FUNCTION_BLOCK DSInterface (* Drill station service interface *)
  (* Standard: 61499-2 *)
  (* Version 0.2, 2003-12-04, JHC, Rockwell Automation, Renamed for better indexing. *)
  (* Version 0.1, 2002-11-05, JHC, Rockwell Automation, Corrected missing ST element in Algorithm REQ. *)
  (* Version 0.0, 2000-05-30, JHC, Rockwell Automation *)
  (* Compiler header: package fb.rt.projects.DrillStation; *)
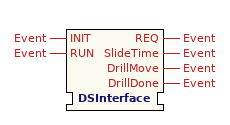
  EVENT_INPUT
    INIT; (* Initialization Request *)
    RUN; (* Run simulation *)
  END_EVENT
  EVENT_OUTPUT
    REQ;
    SlideTime;
    DrillMove;
    DrillDone;
  END_EVENT
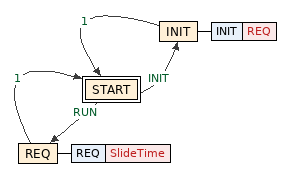
  EC_STATES
    START; (* Initial State *)
    INIT : INIT -> REQ; (* Initialization *)
    REQ : REQ -> SlideTime; (* Normal execution *)
  END_STATES
  EC_TRANSITIONS
    START TO INIT := INIT;
    INIT TO START := 1;
    START TO REQ := RUN;
    REQ TO START := 1;
  END_TRANSITIONS
  ALGORITHM INIT IN Java: (* Initialization algorithm *)
// Interface initialization method
  END_ALGORITHM
  ALGORITHM REQ IN Java: (* Normally executed algorithm *)
// Run the simulation here
  END_ALGORITHM
END_FUNCTION_BLOCK
